// TwinCAT 3 PLC project TcAssignment_4PLC
// ProgramVersion: 3.1.4024.0
// libraries:
//   Tc2_Standard, * (Beckhoff Automation GmbH)
//   Tc2_System, * (Beckhoff Automation GmbH)
//   Tc3_Module, * (Beckhoff Automation GmbH)
// project tree:
//   DUTs/ E_MachineMode.TcDUT, E_MachineState.TcDUT
//   GVLs/ GVL.TcGVL (not stored)
//   / PlcTask.TcTTO
//   POUs/ FB_BottleCounter.TcPOU (not stored), FB_BottleFillingMachine.TcPOU (not stored), FB_Conveyor.TcPOU, FB_FillingUnit.TcPOU (not stored), I_FillingMachine.TcIO (not stored), MAIN.TcPOU (not stored)
// real-time tasks:
//   TASK PlcTask: cycle T#10ms, priority 20, ADS port 350

CONFIGURATION TcAssignment_4PLC
    RESOURCE PLC ON TwinCAT3
        TASK PlcTask(INTERVAL := T#10ms, PRIORITY := 20);
        PROGRAM MAIN WITH PlcTask : MAIN;
    END_RESOURCE
END_CONFIGURATION

// ---- DUTs/E_MachineMode.TcDUT
TYPE E_MachineMode :
(
	auto,
	manual,
	none
);
END_TYPE

// ---- DUTs/E_MachineState.TcDUT
TYPE E_MachineState :
(
    Idle,
    Running,
    Filling,
    Capping,
    Stopped

);
END_TYPE

// ---- POUs/FB_Conveyor.TcPOU
FUNCTION_BLOCK FB_Conveyor
VAR
    bConveyorRunning : BOOL;
END_VAR

GVL.g_bConveyorMotor := bConveyorRunning;

METHOD Start
 bConveyorRunning := TRUE;
END_METHOD

METHOD Stop
 bConveyorRunning := FALSE;
END_METHOD

END_FUNCTION_BLOCK
